SUBAPPLICATION ACTION_SERVER_SEND_GOAL
  (* Standard: 61499-2 *)
  (* Version 1.0, 2023-04-02, Tim Hesse *)
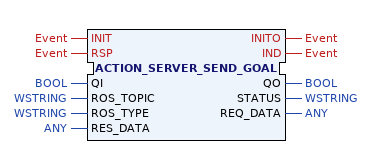
  EVENT_INPUT
    INIT; (* Initialization Request *)
    RSP;
  END_EVENT
  EVENT_OUTPUT
    INITO; (* Initialization Confirm *)
    IND;
  END_EVENT
  VAR_INPUT
    QI : BOOL; (* Input event qualifier *)
    ROS_TOPIC : WSTRING;
    ROS_TYPE : WSTRING;
    RES_DATA : ANY;
  END_VAR
  VAR_OUTPUT
    QO : BOOL; (* Output event qualifier *)
    STATUS : WSTRING;
    REQ_DATA : ANY;
  END_VAR
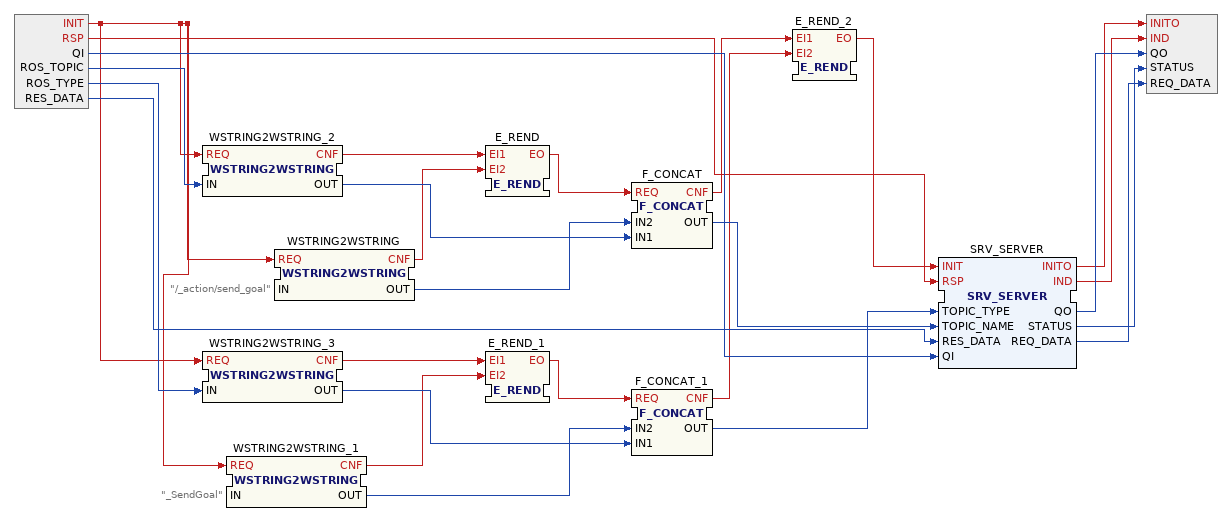
  FBS
    F_CONCAT_1 : F_CONCAT;
    WSTRING2WSTRING_1 : WSTRING2WSTRING(IN := "_SendGoal");
    F_CONCAT : F_CONCAT;
    WSTRING2WSTRING : WSTRING2WSTRING(IN := "/_action/send_goal");
    WSTRING2WSTRING_2 : WSTRING2WSTRING;
    E_REND : E_REND;
    E_REND_1 : E_REND;
    E_REND_2 : E_REND;
    WSTRING2WSTRING_3 : WSTRING2WSTRING;
  END_FBS
  SUBAPPS
    SRV_SERVER : SRV_SERVER;
  END_SUBAPPS
  EVENT_CONNECTIONS
    WSTRING2WSTRING_3.CNF TO E_REND_1.EI1;
    E_REND_1.EO TO F_CONCAT_1.REQ;
    WSTRING2WSTRING_2.CNF TO E_REND.EI1;
    E_REND.EO TO F_CONCAT.REQ;
    WSTRING2WSTRING_1.CNF TO E_REND_1.EI2;
    F_CONCAT.CNF TO E_REND_2.EI1;
    F_CONCAT_1.CNF TO E_REND_2.EI2;
    WSTRING2WSTRING.CNF TO E_REND.EI2;
    E_REND_2.EO TO SRV_SERVER.INIT;
    SRV_SERVER.INITO TO INITO;
    SRV_SERVER.IND TO IND;
    INIT TO WSTRING2WSTRING_2.REQ;
    INIT TO WSTRING2WSTRING.REQ;
    INIT TO WSTRING2WSTRING_3.REQ;
    INIT TO WSTRING2WSTRING_1.REQ;
    RSP TO SRV_SERVER.RSP;
  END_CONNECTIONS
  DATA_CONNECTIONS
    WSTRING2WSTRING.OUT TO F_CONCAT.IN2;
    WSTRING2WSTRING_1.OUT TO F_CONCAT_1.IN2;
    WSTRING2WSTRING_3.OUT TO F_CONCAT_1.IN1;
    WSTRING2WSTRING_2.OUT TO F_CONCAT.IN1;
    F_CONCAT_1.OUT TO SRV_SERVER.TOPIC_TYPE;
    F_CONCAT.OUT TO SRV_SERVER.TOPIC_NAME;
    SRV_SERVER.QO TO QO;
    SRV_SERVER.STATUS TO STATUS;
    SRV_SERVER.REQ_DATA TO REQ_DATA;
    ROS_TOPIC TO WSTRING2WSTRING_2.IN;
    ROS_TYPE TO WSTRING2WSTRING_3.IN;
    RES_DATA TO SRV_SERVER.RES_DATA;
    QI TO SRV_SERVER.QI;
  END_CONNECTIONS
END_SUBAPPLICATION
